# EPICS autosave request: mcaApp/Db/icb_adc_settings.req
# FILE... icb_adc_settings.req
# USAGE.. icb_adc.db fields autosave'd.
$(P)$(ADC)GAIN
$(P)$(ADC)OFFSET
$(P)$(ADC)ULD
$(P)$(ADC)LLD
$(P)$(ADC)ZERO
$(P)$(ADC)PMOD
$(P)$(ADC)GMOD
$(P)$(ADC)TMOD
$(P)$(ADC)CMOD
$(P)$(ADC)AMOD
